FUNCTION Convert_ULINT_TO_DATE : BOOL
VAR_INPUT
	in : ULINT;
	out : REFERENCE TO DATE;
END_VAR
VAR
	converted : DATE;
END_VAR

converted := ULINT_TO_DATE(in);

IF (DATE_TO_ULINT(converted) <> in) THEN
	RETURN;
END_IF

out := converted;
Convert_ULINT_TO_DATE := TRUE;

END_FUNCTION

(* stored: Version 1.1.0.1, ProductVersion 3.1.4024.12
   POU Convert_ULINT_TO_DATE: Id {418fe3e2-f589-4366-8176-480e526f917c}, SpecialFunc None *)
